FUNCTION_BLOCK BB
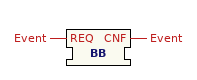
  EVENT_INPUT
    REQ;
  END_EVENT
  EVENT_OUTPUT
    CNF;
  END_EVENT
  VAR
    INTERNALVAR1 : BOOL := FALSE;
  END_VAR
  EC_STATES
    START;
  END_STATES
END_FUNCTION_BLOCK
